// TwinCAT 3 PLC project main
// ProgramVersion: 3.1.4024.0
// libraries:
//   Tc2_Standard, * (Beckhoff Automation GmbH)
//   Tc2_System, * (Beckhoff Automation GmbH)
//   Tc2_Utilities, * (Beckhoff Automation GmbH)
//   Tc3_Module, * (Beckhoff Automation GmbH)
// project tree:
//   DUTs/ E_EventType.TcDUT, ST_Event.TcDUT
//   / PlcTask.TcTTO
//   POUs/ FB_EventRingBuffer.TcPOU, EventStorage.TcIO, FB_EventLogger.TcPOU, FB_CSVEventStorage.TcPOU, F_SystemTimeToDT.TcPOU, F_UpdateEventTimeStamp.TcPOU, MAIN.TcPOU
// real-time tasks:
//   TASK PlcTask: cycle T#10ms, priority 20, ADS port 350

CONFIGURATION main
    RESOURCE PLC ON TwinCAT3
        TASK PlcTask(INTERVAL := T#10ms, PRIORITY := 20);
        PROGRAM MAIN WITH PlcTask : MAIN;
    END_RESOURCE
END_CONFIGURATION

// ---- DUTs/E_EventType.TcDUT
{attribute 'qualified_only'}
{attribute 'strict'}
{attribute 'to_string'}
TYPE E_EventType :
(
	alarm,
	message
);
END_TYPE

// ---- DUTs/ST_Event.TcDUT
TYPE ST_Event :
STRUCT
	eEventType: E_EventType;
	eEventSeverity: TcEventSeverity;
	nEventId: UINT;
	sEventText: STRING(255); // 255 is a good size because most of the twincat built in functions can handle 255
	dtTimeStamp: DATE_AND_TIME;
END_STRUCT
END_TYPE

// ---- POUs/EventStorage.TcIO
INTERFACE EventStorage

METHOD StoreEvent
VAR_INPUT
	st_event: ST_Event;
END_VAR
END_METHOD

END_INTERFACE

// ---- POUs/MAIN.TcPOU
PROGRAM MAIN
VAR
	st_event: ST_Event; // Only this structs copy is being used everywhere.
	once: BOOL := FALSE;
	
	csvEventStorage: FB_CSVEventStorage;
	eventLogger : FB_EventLogger(csvEventStorage);
	
	eventCounter: UINT := 0;
	bIsError : BOOL;
	
	bReadAndRemoveFromBuffer: BOOL;
	lastReadSTEvent: ST_Event;
	nNoOfEventsRemaining: UDINT;
END_VAR

IF once THEN
	st_event.eEventType := E_EventType.alarm;
	st_event.eEventSeverity := TcEventSeverity.Critical;
	st_event.sEventText :=  'This is an event text';
	eventCounter := eventCounter + 1;
	st_event.nEventId := eventCounter;
	
	bIsError := eventLogger.AddEvent(st_event);
	once := FALSE;
END_IF

csvEventStorage();

(*IF NOT once THEN
	F_UpdateEventTimeStamp(st_event:= st_event);
	once := TRUE;
END_IF
*)

END_PROGRAM

// ---- POUs/FB_CSVEventStorage.TcPOU
FUNCTION_BLOCK FB_CSVEventStorage IMPLEMENTS EventStorage
VAR 
	// Enum for state machine
	eWriteState: (	FILE_OPEN_TRIGGER,FILE_OPEN,WAIT_FOR_EVENT,WRITE_EVENT_TRIGGER,
					WRITE_EVENT,FILE_CLOSE_TRIGGER, FILE_CLOSE,ERROR);
				 
	fbFileOpen: FB_FileOpen := (bExecute := FALSE, sPathName := 'C:\Events.log', nMode := FOPEN_MODEAPPEND OR FOPEN_MODETEXT);
	
	fbFilePuts: FB_FilePuts();
	fbFileClose: FB_FileClose();

	stWriteEvent: ST_EVENT; // The st_event which is supposed to be written	
	csvString: T_MaxString;
END_VAR

CASE eWriteState OF
	
	FILE_OPEN_TRIGGER :
		// Start the function, the rising edge is started and the function will be continously called 
		// until windows allows it to be opened
		fbFileOpen(bExecute:= TRUE);
		eWriteState := FILE_OPEN;
		
	FILE_OPEN :
		fbFileOpen(bExecute:= FALSE);
		IF fbFileOpen.bError THEN
			eWriteState := ERROR; // You can also do something like rerunning the above to check again
		ELSIF NOT fbFileOpen.bBusy AND fbFileOpen.hFile <> 0 THEN
			 eWriteState := WAIT_FOR_EVENT;
		END_IF
	
	WAIT_FOR_EVENT :
		// Do Nothing here see StoreEvent
	
	WRITE_EVENT_TRIGGER:
		csvString := STEventToCSVString(stEvent := stWriteEvent);
		fbFilePuts(bExecute:= FALSE);
		fbFilePuts(bExecute:= TRUE, sLine := csvString, hFile := fbFileOpen.hFile);
		eWriteState := WRITE_EVENT;
	
	WRITE_EVENT :
		fbFilePuts(bExecute:= FALSE);
		IF fbFilePuts.bError THEN
			eWriteState := Error;
		ELSIF NOT fbFilePuts.bBusy THEN
			// This was for when we had to coninously wait for new writes in storeEVent method
			// But it wouldn't write as the file had to be closed
			// eWriteState:= WAIT_FOR_EVENT; 
			
			eWriteState:= FILE_CLOSE_TRIGGER;
		END_IF
		
	
	FILE_CLOSE_TRIGGER: 
		fbFileClose(bExecute := FALSE);
		fbFileClose(bExecute := TRUE, hFile :=fbFileOpen.hFile);
		eWriteState := FILE_CLOSE;
		
	FILE_CLOSE :
		fbFileClose(bExecute := FALSE);
		IF fbFileClose.bError THEN
			eWriteState := Error;
		ELSIF NOT fbFileClose.bBusy THEN
			eWriteState := FILE_OPEN_TRIGGER;
		END_IF
	
	ERROR :
		fbFileOpen.nErrId;
	
END_CASE

METHOD PRIVATE STEventToCSVString: T_MaxString
VAR_INPUT
	stEvent : REFERENCE TO ST_EVENT;
END_VAR
VAR
	stringHolder: T_MaxString;
END_VAR
stringHolder := TO_STRING(stEvent.eEventType); // This works because of the attribute added to the enum
stringHolder := CONCAT(str1 := stringHolder, str2 := ',');

stringHolder := CONCAT(str1 := stringHolder, str2 := TO_STRING(stEvent.eEventSeverity)); // Here only numbers will be added
stringHolder := CONCAT(str1 := stringHolder, str2 := ',');

stringHolder := CONCAT(str1 := stringHolder, str2 := TO_STRING(stEvent.nEventId));
stringHolder := CONCAT(str1 := stringHolder, str2 := ',');

stringHolder := CONCAT(str1 := stringHolder, str2 := F_RTRIM(stEvent.sEventText));
stringHolder := CONCAT(str1 := stringHolder, str2 := ',');

stringHolder := CONCAT(str1 := stringHolder, str2 := TO_STRING(stEvent.dtTimeStamp));
stringHolder := CONCAT(str1 := stringHolder, str2 := '$n'); // New line

STEventToCSVString := stringHolder;
END_METHOD

// add method implementation 
METHOD StoreEvent
VAR_INPUT
	st_event	: ST_Event;
END_VAR
IF eWriteState = WAIT_FOR_EVENT THEN
	eWriteState := WRITE_EVENT_TRIGGER;
	stWriteEvent:= st_event;
END_IF
END_METHOD

END_FUNCTION_BLOCK

// ---- POUs/FB_EventLogger.TcPOU
FUNCTION_BLOCK FB_EventLogger
VAR
	eventBuffer: ARRAY[1..EVENT_BUFFER_SIZE] OF ST_Event;
	currentBufferIndex: USINT := 0;
	
	_eventStorage: EventStorage; // setting this in the constructor/FB_init
	ringBuffer: FB_EventRingBuffer;
	
END_VAR
VAR CONSTANT
	EVENT_BUFFER_SIZE: INT := 10;
END_VAR

METHOD AddEvent : BOOL
VAR_INPUT
	event: ST_EVENT;
	// event: REFERENCE TO ST_EVENT;
END_VAR
VAR
	readEvent: ST_EVENT;
	bIsReadFailed: BOOL;
	nRemainingEventCount: UDINT;
END_VAR
(*
IF (currentBufferIndex + 1) < EVENT_BUFFER_SIZE THEN
	currentBufferIndex := currentBufferIndex + 1;
	F_UpdateEventTimeStamp(st_event := event);
	event.nEventId := currentBufferIndex;

	eventBuffer[currentBufferIndex]:= event;
	
	// Here we store event persistently
	_eventStorage.StoreEvent(st_event:= event);
END_IF 
*)

// Using the RingBuffer here
F_UpdateEventTimeStamp(st_event := event);
ringBuffer.AddEvent(stEvent:= event, bIsError => AddEvent);


// Here we store event persistently
//_eventStorage.StoreEvent(st_event:= event);
IF ringBuffer.GetBufferEventCount() > 0 THEN
	ringBuffer.GetAndRemoveEvent(stEvent => readEvent, bError => bIsReadFailed);
	_eventStorage.StoreEvent(readEvent);	
END_IF
END_METHOD

(****
 
Called implicitly whenever an instance of the Event Logger is instantiated.
Like a Constructor.

*****)

METHOD FB_init : BOOL
VAR_INPUT
	bInitRetains : BOOL; // if TRUE, the retain variables are initialized (warm start / cold start)
	bInCopyCode : BOOL;  // if TRUE, the instance afterwards gets moved into the copy code (online change)

	// Require something that implementes EventStorage interface	
	eventStorage: EventStorage;
	
END_VAR
_eventStorage := eventStorage;
END_METHOD

END_FUNCTION_BLOCK

// ---- POUs/FB_EventRingBuffer.TcPOU
FUNCTION_BLOCK FB_EventRingBuffer
VAR
	ringBuffer: FB_MemRingBuffer;
	arrBuffer : ARRAY[0..MAX_BUFFER_SIZE] OF BYTE; (*Buffer memory used by the FB_MemRingBuffer*)
END_VAR
VAR CONSTANT
	SIZE_OF_ST_EVENT: UDINT := SIZEOF(ST_Event); // Get the number of bytes required for ST_EVENT
	MAX_NUM_OF_ST_EVENTS: UDINT := 5;
	
	// Now the ring buffer size to store 5 ST_EVENTS
	MAX_BUFFER_SIZE: UDINT := SIZE_OF_ST_EVENT * MAX_NUM_OF_ST_EVENTS;
END_VAR

METHOD AddEvent
VAR_INPUT
	stEvent: REFERENCE TO ST_Event;
END_VAR
VAR_OUTPUT
	bIsError: Bool;
END_VAR
ringBuffer.A_AddTail(
	pWrite := ADR(stEvent),
	cbWrite:= SIZEOF(stEvent),
	pBuffer:= ADR(arrBuffer),
	cbBuffer:= SIZEOF(arrBuffer)
);

// Returns TRUE, if a new data set was added or removed successfully.
// Returns FALSE in the event of a buffer overflow or if no more entries are available in the buffer.
bIsError := NOT ringBuffer.bOk;
END_METHOD

METHOD ClearRingBuffer : BOOL
ringBuffer.A_Reset(
	pBuffer:= ADR(arrBuffer),
	cbBuffer:= SIZEOF(arrBuffer)
);

ClearRingBuffer := ringBuffer.bOk;
END_METHOD

METHOD GetAndRemoveEvent
VAR_OUTPUT
	stEvent: ST_Event;
	bError: BOOL;
END_VAR
ringBuffer.A_RemoveHead(
	pRead := ADR(stEvent),
	cbRead:= SIZEOF(stEvent),
	pBuffer:= ADR(arrBuffer),
	cbBuffer:= SIZEOF(arrBuffer)
);

bError := NOT ringBuffer.bOk;
END_METHOD

METHOD GetBufferEventCount : UDINT
GetBufferEventCount :=	ringBuffer.nCount;
END_METHOD

END_FUNCTION_BLOCK

// ---- POUs/F_UpdateEventTimeStamp.TcPOU
FUNCTION F_UpdateEventTimeStamp
VAR_INPUT
	st_event : REFERENCE TO ST_Event;
END_VAR
VAR
	ulns: ULINT;
	fileTime: T_FILETIME;
END_VAR

ulns := F_GETSYSTEMTIME();
st_event.dtTimeStamp := F_SystemTimeToDT(nSystemTime:= ulns);

END_FUNCTION

// ---- POUs/F_SystemTimeToDT.TcPOU
FUNCTION F_SystemTimeToDT : DT
VAR CONSTANT
    SECONDS_BETWEEN_1601_AND_1970 : ULINT := 11_644_473_600;
END_VAR
VAR_INPUT
    nSystemTime : ULINT; // One unit is 100 ns since 1 January 1601
END_VAR
VAR
    nSeconds : ULINT;
END_VAR

// Unix time is measured in seconds since January 1, 1970.
nSeconds := (nSystemTime / 10_000_000) - SECONDS_BETWEEN_1601_AND_1970;
F_SystemTimeToDT := ULINT_TO_DT(nSeconds); // It is returning it in UTC

END_FUNCTION
